Staubli VAL3: bool2num.pgx

public program bool2num(bool& x_bInput[], num& x_nResult[], bool& x_bError)
  local num l_nLength
  local num l_nElement
begin

  x_bError = false
  l_nLength = size(x_bInput)
  x_nResult = 0
  resize(x_nResult, 1, l_nLength)

  for l_nElement = 0 to l_nLength-1
    if x_bInput[l_nElement] == true
      x_nResult[l_nElement] = 1
    elseIf x_bInput[l_nElement] == false
      x_nResult[l_nElement] = 0
    else
      x_bError = true
    endIf
  endFor

end
